FUNCTION_BLOCK MERGE
  {SET_ATTRIBUTE(OpcUa, SERVICE)}
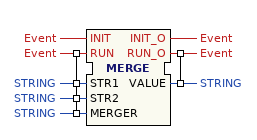
  EVENT_INPUT
    INIT;
    RUN WITH STR1, STR2, MERGER;
  END_EVENT
  EVENT_OUTPUT
    INIT_O;
    RUN_O WITH VALUE;
  END_EVENT
  VAR_INPUT
    STR1 : STRING; {SET_ATTRIBUTE(OpcUa, Variable)}
    STR2 : STRING; {SET_ATTRIBUTE(OpcUa, Variable)}
    MERGER : STRING; {SET_ATTRIBUTE(OpcUa, Constant)}
  END_VAR
  VAR_OUTPUT
    VALUE : STRING; {SET_ATTRIBUTE(OpcUa, Variable)}
  END_VAR
END_FUNCTION_BLOCK
